ABB RobotStudio station: task2_Diaz_Raphael_good.rsstn

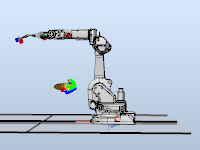
Station task2_Diaz_Raphael_good (saved by RobotStudio 7.0.8732.594)
Controller IRB_1660ID_4kg_1.55m_1
  mechanical unit ROB_1: IRB1660ID_4_155__03, 6 joints, base frame (0, 0, 0) mm
Layout (positions relative to the parent item):
  - IRB1660ID_4_155__03 [mechanism, from Robots\IRB1660ID_4_155__03.rslib] at (0, 0, 0) mm; joint values [0, 0, 0, 0, 0, 0] (rad or m)
  - Binzel_ID_22 [mechanism, from Tools\Binzel_ID_22.rslib] at (962.96, 0, 1296.5) mm, rotated rx 0 ry 90 rz 0 deg
  - propeller [part, from Training Objects\propeller.rslib] at (600, 300, 492) mm
Attachment: Binzel_ID_22 is attached to IRB1660ID_4_155__03 / Link6
Collision set Jeu de collisions_1: propeller against Binzel_ID_22, near miss 0.01 m
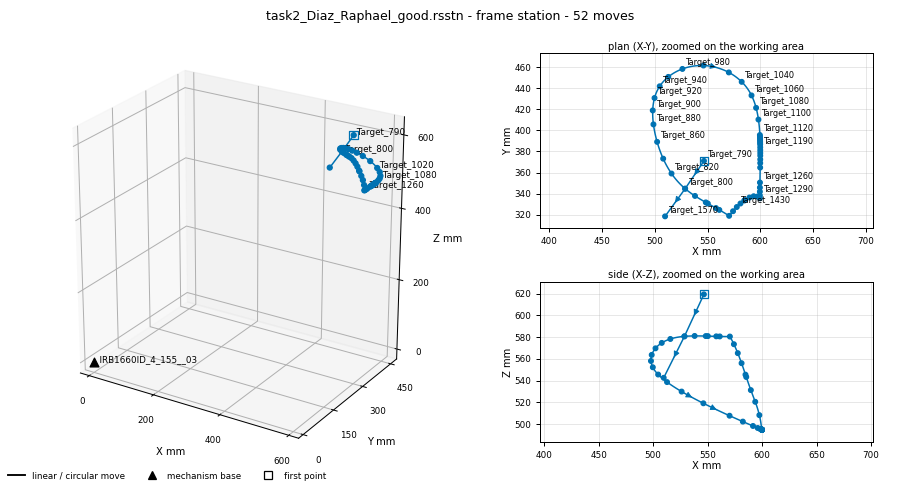
[picture p0: tool path of task2_Diaz_Raphael_good.rsstn in frame station, 52 of 54 moves have a stored position in this frame; points joined in program order, loops and branches not executed]
Targets, tools, work objects and paths stored in the station, written as RAPID:
! task T_ROB1
MODULE CalibData
  PERS tooldata tWeldGun:=[TRUE,[[49.841566361,0,372.194826196],[0.981627183,0,0.190808995,0]],[2,[0,0,100],[0,1,0,0],0,0,0]];
  TASK PERS wobjdata wobjpropeller:=[FALSE,TRUE,"",[[600,300,492],[1,0,0,0]],[[0,0,0],[1,0,0,0]]];
ENDMODULE

! task T_ROB1
MODULE Module1
  CONST robtarget Target_10:=[[-91.457935103,19.381495894,50.577643768],[0.33610531,0.650809481,-0.678295692,0.058268297],[0,0,0,0],[9E+09,9E+09,9E+09,9E+09,9E+09,9E+09]];
  CONST robtarget Target_20:=[[-71.308296548,44.654165227,88.72583181],[0.299329258,0.383053383,-0.856704989,0.172420021],[0,0,0,0],[9E+09,9E+09,9E+09,9E+09,9E+09,9E+09]];
  CONST robtarget Target_30:=[[-78.37226907,51.547933238,87.786349051],[0.117055584,0.822479759,0.470472306,-0.297457301],[0,0,0,0],[9E+09,9E+09,9E+09,9E+09,9E+09,9E+09]];
  CONST robtarget Target_40:=[[-84.2413284,59.034723416,86.319213476],[0.026567482,0.682501524,0.663067393,-0.306312701],[0,0,0,0],[9E+09,9E+09,9E+09,9E+09,9E+09,9E+09]];
  CONST robtarget Target_50:=[[-88.689736644,66.246127572,84.593004406],[0.015778406,-0.605999209,-0.736035915,0.301275841],[0,0,0,0],[9E+09,9E+09,9E+09,9E+09,9E+09,9E+09]];
  CONST robtarget Target_60:=[[-92.125721625,73.134318692,82.720919892],[0.04515113,-0.547999882,-0.781238502,0.29550619],[0,0,0,0],[9E+09,9E+09,9E+09,9E+09,9E+09,9E+09]];
  CONST robtarget Target_70:=[[-95.368783045,81.204603576,80.298199397],[0.073925684,-0.486542001,-0.821345688,0.288449537],[0,0,0,0],[9E+09,9E+09,9E+09,9E+09,9E+09,9E+09]];
  CONST robtarget Target_80:=[[-97.881197354,89.077633701,77.728399267],[0.099335356,-0.428105921,-0.853147584,0.281064062],[0,0,0,0],[9E+09,9E+09,9E+09,9E+09,9E+09,9E+09]];
  CONST robtarget Target_90:=[[-100.033550677,97.806160497,74.661081462],[0.123258623,-0.370832778,-0.879360143,0.272059003],[0,0,0,0],[9E+09,9E+09,9E+09,9E+09,9E+09,9E+09]];
  CONST robtarget Target_100:=[[-101.370571802,105.645030719,71.694531974],[0.137199941,-0.339206789,-0.892353586,0.264234759],[0,0,0,0],[9E+09,9E+09,9E+09,9E+09,9E+09,9E+09]];
  CONST robtarget Target_110:=[[-101.985517598,112.196954226,69.035342228],[0.143656337,-0.327575869,-0.897345121,0.25851236],[0,0,0,0],[9E+09,9E+09,9E+09,9E+09,9E+09,9E+09]];
  CONST robtarget Target_120:=[[-102.050783732,118.905008267,66.110246882],[0.145775207,-0.329044052,-0.897889581,0.253522978],[0,0,0,0],[9E+09,9E+09,9E+09,9E+09,9E+09,9E+09]];
  CONST robtarget Target_130:=[[-101.533339164,124.816905053,63.325398927],[0.144182461,-0.340855073,-0.894813654,0.249675314],[0,0,0,0],[9E+09,9E+09,9E+09,9E+09,9E+09,9E+09]];
  CONST robtarget Target_140:=[[-100.353288111,130.675770651,60.324888075],[0.139634307,-0.361631976,-0.888364776,0.246033736],[0,0,0,0],[9E+09,9E+09,9E+09,9E+09,9E+09,9E+09]];
  CONST robtarget Target_150:=[[-98.373944468,136.376977106,57.10491509],[0.132520307,-0.390029479,-0.878439143,0.242198359],[0,0,0,0],[9E+09,9E+09,9E+09,9E+09,9E+09,9E+09]];
  CONST robtarget Target_160:=[[-95.443552762,141.799075074,53.663228181],[0.123926919,-0.422628209,-0.865746717,0.23771861],[0,0,0,0],[9E+09,9E+09,9E+09,9E+09,9E+09,9E+09]];
  CONST robtarget Target_170:=[[-91.477533598,146.819277823,50.007346793],[0.119671198,-0.442406606,-0.857808795,0.232635489],[0,0,0,0],[9E+09,9E+09,9E+09,9E+09,9E+09,9E+09]];
  CONST robtarget Target_180:=[[-87.281413645,150.715782558,46.72049795],[0.119661723,-0.448819982,-0.855661661,0.228220987],[0,0,0,0],[9E+09,9E+09,9E+09,9E+09,9E+09,9E+09]];
  CONST robtarget Target_190:=[[-80.620544648,155.184469083,42.151881558],[0.123978964,-0.4449886,-0.858578449,0.222390219],[0,0,0,0],[9E+09,9E+09,9E+09,9E+09,9E+09,9E+09]];
  CONST robtarget Target_200:=[[-73.893581114,158.264895339,38.018756325],[0.131604396,-0.430683265,-0.866049681,0.217140869],[0,0,0,0],[9E+09,9E+09,9E+09,9E+09,9E+09,9E+09]];
  CONST robtarget Target_210:=[[-64.220289368,160.829182326,32.592775118],[0.147131247,-0.395863657,-0.88192952,0.209391221],[0,0,0,0],[9E+09,9E+09,9E+09,9E+09,9E+09,9E+09]];
  CONST robtarget Target_220:=[[-53.911152598,161.491173917,27.246893168],[0.169941176,-0.339310055,-0.903559757,0.198918197],[0,0,0,0],[9E+09,9E+09,9E+09,9E+09,9E+09,9E+09]];
  CONST robtarget Target_230:=[[-41.810424561,159.659563045,21.355681333],[0.200569217,-0.259415196,-0.927008519,0.182019097],[0,0,0,0],[9E+09,9E+09,9E+09,9E+09,9E+09,9E+09]];
  CONST robtarget Target_240:=[[-29.865399659,154.942077691,15.837356936],[0.23576805,-0.163069983,-0.945025663,0.157315299],[0,0,0,0],[9E+09,9E+09,9E+09,9E+09,9E+09,9E+09]];
  CONST robtarget Target_250:=[[-23.746821381,151.136846643,13.101781769],[0.258743132,-0.097071717,-0.951106966,0.137929734],[0,0,0,0],[9E+09,9E+09,9E+09,9E+09,9E+09,9E+09]];
  CONST robtarget Target_260:=[[-17.666404877,146.023270878,10.434303465],[0.288578567,-0.007433268,-0.951293254,0.108204906],[0,0,0,0],[9E+09,9E+09,9E+09,9E+09,9E+09,9E+09]];
  CONST robtarget Target_270:=[[-12.651720819,140.244931337,8.266059989],[0.323388208,0.102706042,-0.938405879,0.065314172],[0,0,0,0],[9E+09,9E+09,9E+09,9E+09,9E+09,9E+09]];
  CONST robtarget Target_280:=[[-8.342471887,133.132300705,6.417634315],[0.365484893,0.241842337,-0.898844698,-0.003359375],[0,0,0,0],[9E+09,9E+09,9E+09,9E+09,9E+09,9E+09]];
  CONST robtarget Target_290:=[[-5.860288763,127.302609884,5.357964601],[0.392577974,0.330559163,-0.856027592,-0.061886481],[0,0,0,0],[9E+09,9E+09,9E+09,9E+09,9E+09,9E+09]];
  CONST robtarget Target_300:=[[-3.992732838,121.340092984,4.564472039],[0.414682372,0.398212956,-0.809177456,-0.12123043],[0,0,0,0],[9E+09,9E+09,9E+09,9E+09,9E+09,9E+09]];
  CONST robtarget Target_310:=[[-2.622802171,115.344004565,3.985624159],[0.432618645,0.446096603,-0.762723965,-0.179139837],[0,0,0,0],[9E+09,9E+09,9E+09,9E+09,9E+09,9E+09]];
  CONST robtarget Target_320:=[[-1.767059875,110.242020204,3.626183876],[0.445232804,0.473650463,-0.725447966,-0.22615976],[0,0,0,0],[9E+09,9E+09,9E+09,9E+09,9E+09,9E+09]];
  CONST robtarget Target_330:=[[-0.982577099,103.57416667,3.298978191],[0.458683869,0.49524232,-0.681313145,-0.283119323],[0,0,0,0],[9E+09,9E+09,9E+09,9E+09,9E+09,9E+09]];
  CONST robtarget Target_340:=[[-0.419164603,95.575819275,3.066095193],[0.470824783,0.505758987,-0.636794178,-0.342089236],[0,0,0,0],[9E+09,9E+09,9E+09,9E+09,9E+09,9E+09]];
  CONST robtarget Target_350:=[[-0.347305784,94.031887162,3.036532706],[0.472698308,0.506466011,-0.629402289,-0.35199609],[0,0,0,0],[9E+09,9E+09,9E+09,9E+09,9E+09,9E+09]];
  CONST robtarget Target_360:=[[-0.286087854,92.508600465,3.011348256],[0.474402212,0.506869723,-0.622525025,-0.361231531],[0,0,0,0],[9E+09,9E+09,9E+09,9E+09,9E+09,9E+09]];
  CONST robtarget Target_370:=[[-0.23439904,91.006691049,2.990058478],[0.475942955,0.507030195,-0.616165129,-0.369782665],[0,0,0,0],[9E+09,9E+09,9E+09,9E+09,9E+09,9E+09]];
  CONST robtarget Target_380:=[[-0.191127564,89.526890776,2.972180009],[0.477327032,0.507002401,-0.610324314,-0.377639647],[0,0,0,0],[9E+09,9E+09,9E+09,9E+09,9E+09,9E+09]];
  CONST robtarget Target_390:=[[-0.155200515,88.069901279,2.957246513],[0.478560799,0.506836069,-0.605003836,-0.384794905],[0,0,0,0],[9E+09,9E+09,9E+09,9E+09,9E+09,9E+09]];
  CONST robtarget Target_400:=[[-0.125712724,86.636254313,2.944866369],[0.47965026,0.506575668,-0.600205327,-0.391241979],[0,0,0,0],[9E+09,9E+09,9E+09,9E+09,9E+09,9E+09]];
  CONST robtarget Target_410:=[[-0.08261427,83.840896172,2.926280967],[0.481425707,0.505921465,-0.592147985,-0.402036719],[0,0,0,0],[9E+09,9E+09,9E+09,9E+09,9E+09,9E+09]];
  CONST robtarget Target_420:=[[-0.056032781,81.142526543,2.913966515],[0.482919894,0.505164577,-0.585071946,-0.411446161],[0,0,0,0],[9E+09,9E+09,9E+09,9E+09,9E+09,9E+09]];
  CONST robtarget Target_430:=[[-0.043048917,78.537720407,2.906816995],[0.484257027,0.504334678,-0.578448423,-0.420165547],[0,0,0,0],[9E+09,9E+09,9E+09,9E+09,9E+09,9E+09]];
  CONST robtarget Target_440:=[[-0.0411167,76.022616297,2.903894485],[0.485444308,0.50348214,-0.572280664,-0.428187343],[0,0,0,0],[9E+09,9E+09,9E+09,9E+09,9E+09,9E+09]];
  CONST robtarget Target_450:=[[-0.054549222,72.411596474,2.905814438],[0.486961818,0.502254961,-0.563882455,-0.43891311],[0,0,0,0],[9E+09,9E+09,9E+09,9E+09,9E+09,9E+09]];
  CONST robtarget Target_460:=[[-0.082166755,68.986528626,2.913297006],[0.488190694,0.501190902,-0.556485739,-0.448108412],[0,0,0,0],[9E+09,9E+09,9E+09,9E+09,9E+09,9E+09]];
  CONST robtarget Target_470:=[[-0.131718126,64.695350259,2.928466957],[0.489437258,0.500158131,-0.54809675,-0.458129859],[0,0,0,0],[9E+09,9E+09,9E+09,9E+09,9E+09,9E+09]];
  CONST robtarget Target_480:=[[-0.336493102,50.490109414,2.996479603],[0.49131632,0.501098619,-0.528226501,-0.478001266],[0,0,0,0],[9E+09,9E+09,9E+09,9E+09,9E+09,9E+09]];
  CONST robtarget Target_490:=[[-0.389538706,45.718395544,3.014646231],[0.491239016,0.503319057,-0.524352335,-0.480009151],[0,0,0,0],[9E+09,9E+09,9E+09,9E+09,9E+09,9E+09]];
  CONST robtarget Target_500:=[[-0.416651037,41.829820629,3.023974096],[0.490943622,0.505849897,-0.522175178,-0.480024296],[0,0,0,0],[9E+09,9E+09,9E+09,9E+09,9E+09,9E+09]];
  CONST robtarget Target_510:=[[-0.425239936,38.15628616,3.026910604],[0.490487838,0.508788687,-0.520869322,-0.478801528],[0,0,0,0],[9E+09,9E+09,9E+09,9E+09,9E+09,9E+09]];
  CONST robtarget Target_520:=[[-0.41907447,35.554875844,3.024714783],[0.490068794,0.511158358,-0.520350237,-0.477268625],[0,0,0,0],[9E+09,9E+09,9E+09,9E+09,9E+09,9E+09]];
  CONST robtarget Target_530:=[[-1.239353828,36.579195021,10.094804089],[0.485285471,0.505393808,-0.570570399,-0.428397631],[0,0,0,0],[9E+09,9E+09,9E+09,9E+09,9E+09,9E+09]];
  CONST robtarget Target_540:=[[-2.503019666,37.269792356,16.365865608],[0.479926257,0.507544354,-0.597699632,-0.393477656],[0,0,0,0],[9E+09,9E+09,9E+09,9E+09,9E+09,9E+09]];
  CONST robtarget Target_550:=[[-4.236986629,37.619005876,22.65445378],[0.472203187,0.526252128,-0.609551252,-0.358510975],[0,0,0,0],[9E+09,9E+09,9E+09,9E+09,9E+09,9E+09]];
  CONST robtarget Target_560:=[[-6.286575332,37.504452968,28.619621674],[0.462621307,0.570105136,-0.592015985,-0.332383415],[0,0,0,0],[9E+09,9E+09,9E+09,9E+09,9E+09,9E+09]];
  CONST robtarget Target_570:=[[-8.20610761,37.063247875,33.701409225],[0.453744324,0.629847272,-0.535614332,-0.332454193],[0,0,0,0],[9E+09,9E+09,9E+09,9E+09,9E+09,9E+09]];
  CONST robtarget Target_580:=[[-10.318626049,36.285780987,39.360011182],[0.4392884,0.703953672,-0.435520626,-0.348993861],[0,0,0,0],[9E+09,9E+09,9E+09,9E+09,9E+09,9E+09]];
  CONST robtarget Target_590:=[[-12.661310127,35.078889502,45.926428415],[0.411372895,0.780339138,-0.279004478,-0.379472886],[0,0,0,0],[9E+09,9E+09,9E+09,9E+09,9E+09,9E+09]];
  CONST robtarget Target_600:=[[-14.532992973,33.887723981,51.407083874],[0.377332955,0.820678051,-0.122575,-0.411196725],[0,0,0,0],[9E+09,9E+09,9E+09,9E+09,9E+09,9E+09]];
  CONST robtarget Target_610:=[[-10.798566102,36.060475375,40.678801419],[0.563334326,0.293280069,-0.772407011,0.005352333],[0,0,-2,0],[9E+09,9E+09,9E+09,9E+09,9E+09,9E+09]];
  CONST robtarget Target_620:=[[-17.018667911,32.078049469,58.829591721],[0.549464464,0.601489484,-0.578324534,-0.042894489],[0,0,0,0],[9E+09,9E+09,9E+09,9E+09,9E+09,9E+09]];
  CONST robtarget Target_630:=[[-18.838902409,30.609710668,64.071754814],[0.530289122,0.699136232,-0.471191576,-0.089333504],[0,0,0,0],[9E+09,9E+09,9E+09,9E+09,9E+09,9E+09]];
  CONST robtarget Target_640:=[[-20.744338327,28.895776947,69.241801524],[0.123477381,0.8147616,-0.542306034,-0.163771293],[0,0,0,0],[9E+09,9E+09,9E+09,9E+09,9E+09,9E+09]];
  CONST robtarget Target_650:=[[-22.309539778,27.279666365,73.303790841],[0.110236403,0.855139822,-0.430096695,-0.267582985],[0,0,0,0],[9E+09,9E+09,9E+09,9E+09,9E+09,9E+09]];
  CONST robtarget Target_660:=[[-23.973327026,25.503693293,77.244247794],[0.470774997,0.638586467,-0.601652731,0.09269422],[0,0,0,0],[9E+09,9E+09,9E+09,9E+09,9E+09,9E+09]];
  CONST robtarget Target_670:=[[-25.872608406,23.295941961,81.501586218],[0.457862129,0.733090582,-0.501721122,0.034876705],[0,0,0,0],[9E+09,9E+09,9E+09,9E+09,9E+09,9E+09]];
  CONST robtarget Target_680:=[[-27.702454631,21.186772281,85.158169778],[0.001522806,-0.45137891,-0.779666651,0.434021512],[0,0,0,0],[9E+09,9E+09,9E+09,9E+09,9E+09,9E+09]];
  CONST robtarget Target_690:=[[-29.579108704,18.917792453,88.550574629],[0.047769483,-0.396812931,-0.828772501,0.391655098],[0,0,0,0],[9E+09,9E+09,9E+09,9E+09,9E+09,9E+09]];
  CONST robtarget Target_700:=[[-34.181159805,21.772283678,88.563733649],[0.00902881,-0.455561574,-0.785071733,0.419576581],[0,0,0,0],[9E+09,9E+09,9E+09,9E+09,9E+09,9E+09]];
  CONST robtarget Target_710:=[[-38.892044155,24.513127262,88.646240796],[0.005175513,0.466142387,0.770169888,-0.435342202],[0,0,0,0],[9E+09,9E+09,9E+09,9E+09,9E+09,9E+09]];
  CONST robtarget Target_720:=[[-42.068819563,26.298976235,88.725674008],[0.008188854,0.465500607,0.767643082,-0.440415969],[0,0,0,0],[9E+09,9E+09,9E+09,9E+09,9E+09,9E+09]];
  CONST robtarget Target_730:=[[-49.791866469,30.580230673,88.941782186],[0.000167691,-0.452797516,-0.778146204,0.435273324],[0,0,0,0],[9E+09,9E+09,9E+09,9E+09,9E+09,9E+09]];
  CONST robtarget Target_740:=[[-51.709318387,31.655936915,88.990570919],[0.0053493,-0.447245007,-0.783953208,0.430535315],[0,0,0,0],[9E+09,9E+09,9E+09,9E+09,9E+09,9E+09]];
  CONST robtarget Target_750:=[[-57.377839054,34.942502242,89.094223182],[0.02849914,-0.420022979,-0.809203176,0.409827666],[0,0,0,0],[9E+09,9E+09,9E+09,9E+09,9E+09,9E+09]];
  CONST robtarget Target_760:=[[-61.957234754,37.792717573,89.103595138],[0.059645275,-0.371858872,-0.84212475,0.385991355],[0,0,0,0],[9E+09,9E+09,9E+09,9E+09,9E+09,9E+09]];
  CONST robtarget Target_770:=[[-66.351329922,40.79265749,89.011564709],[0.115406616,-0.253755157,-0.893913867,0.351009446],[0,0,0,0],[9E+09,9E+09,9E+09,9E+09,9E+09,9E+09]];
  CONST robtarget Target_780:=[[-71.308296548,44.654165227,88.72583181],[0.299329258,0.383053383,-0.856704989,0.172420021],[0,0,0,0],[9E+09,9E+09,9E+09,9E+09,9E+09,9E+09]];
  CONST robtarget Target_790:=[[-53.446490384,71.034227347,127.305248995],[0.33610531,0.650809481,-0.678295692,0.058268297],[0,0,0,0],[9E+09,9E+09,9E+09,9E+09,9E+09,9E+09]];
  CONST robtarget Target_800:=[[-71.308296548,44.654165227,88.72583181],[0.33610531,0.650809481,-0.678295692,0.058268297],[0,0,0,0],[9E+09,9E+09,9E+09,9E+09,9E+09,9E+09]];
  CONST robtarget Target_810:=[[-78.37226907,51.547933238,87.786349051],[0.33610531,0.650809481,-0.678295692,0.058268297],[0,0,0,0],[9E+09,9E+09,9E+09,9E+09,9E+09,9E+09]];
  CONST robtarget Target_820:=[[-84.2413284,59.034723416,86.319213476],[0.33610531,0.650809481,-0.678295692,0.058268297],[0,0,0,0],[9E+09,9E+09,9E+09,9E+09,9E+09,9E+09]];
  CONST robtarget Target_830:=[[-88.689736644,66.246127572,84.593004406],[0.33610531,0.650809481,-0.678295692,0.058268297],[0,0,0,0],[9E+09,9E+09,9E+09,9E+09,9E+09,9E+09]];
  CONST robtarget Target_840:=[[-92.125721625,73.134318692,82.720919892],[0.33610531,0.650809481,-0.678295692,0.058268297],[0,0,0,0],[9E+09,9E+09,9E+09,9E+09,9E+09,9E+09]];
  CONST robtarget Target_850:=[[-95.368783045,81.204603576,80.298199397],[0.33610531,0.650809481,-0.678295692,0.058268297],[0,0,0,0],[9E+09,9E+09,9E+09,9E+09,9E+09,9E+09]];
  CONST robtarget Target_860:=[[-97.881197354,89.077633701,77.728399267],[0.33610531,0.650809481,-0.678295692,0.058268297],[0,0,0,0],[9E+09,9E+09,9E+09,9E+09,9E+09,9E+09]];
  CONST robtarget Target_870:=[[-100.033550677,97.806160497,74.661081462],[0.33610531,0.650809481,-0.678295692,0.058268297],[0,0,0,0],[9E+09,9E+09,9E+09,9E+09,9E+09,9E+09]];
  CONST robtarget Target_880:=[[-101.370571802,105.645030719,71.694531974],[0.33610531,0.650809481,-0.678295692,0.058268297],[0,0,0,0],[9E+09,9E+09,9E+09,9E+09,9E+09,9E+09]];
  CONST robtarget Target_890:=[[-101.985517598,112.196954226,69.035342228],[0.33610531,0.650809481,-0.678295692,0.058268297],[0,0,0,0],[9E+09,9E+09,9E+09,9E+09,9E+09,9E+09]];
  CONST robtarget Target_900:=[[-102.050783732,118.905008267,66.110246882],[0.33610531,0.650809481,-0.678295692,0.058268297],[0,0,0,0],[9E+09,9E+09,9E+09,9E+09,9E+09,9E+09]];
  CONST robtarget Target_910:=[[-101.533339164,124.816905053,63.325398927],[0.33610531,0.650809481,-0.678295692,0.058268297],[0,0,0,0],[9E+09,9E+09,9E+09,9E+09,9E+09,9E+09]];
  CONST robtarget Target_920:=[[-100.353288111,130.675770651,60.324888075],[0.33610531,0.650809481,-0.678295692,0.058268297],[0,0,0,0],[9E+09,9E+09,9E+09,9E+09,9E+09,9E+09]];
  CONST robtarget Target_930:=[[-98.373944468,136.376977106,57.10491509],[0.33610531,0.650809481,-0.678295692,0.058268297],[0,0,0,0],[9E+09,9E+09,9E+09,9E+09,9E+09,9E+09]];
  CONST robtarget Target_940:=[[-95.443552762,141.799075074,53.663228181],[0.33610531,0.650809481,-0.678295692,0.058268297],[0,0,0,0],[9E+09,9E+09,9E+09,9E+09,9E+09,9E+09]];
  CONST robtarget Target_950:=[[-91.477533598,146.819277823,50.007346793],[0.33610531,0.650809481,-0.678295692,0.058268297],[0,0,0,0],[9E+09,9E+09,9E+09,9E+09,9E+09,9E+09]];
  CONST robtarget Target_960:=[[-87.281413645,150.715782558,46.72049795],[0.33610531,0.650809481,-0.678295692,0.058268297],[0,0,0,0],[9E+09,9E+09,9E+09,9E+09,9E+09,9E+09]];
  CONST robtarget Target_970:=[[-80.620544648,155.184469083,42.151881558],[0.33610531,0.650809481,-0.678295692,0.058268297],[0,0,0,0],[9E+09,9E+09,9E+09,9E+09,9E+09,9E+09]];
  CONST robtarget Target_980:=[[-73.893581114,158.264895339,38.018756325],[0.33610531,0.650809481,-0.678295692,0.058268297],[0,0,0,0],[9E+09,9E+09,9E+09,9E+09,9E+09,9E+09]];
  CONST robtarget Target_990:=[[-64.220289368,160.829182326,32.592775118],[0.33610531,0.650809481,-0.678295692,0.058268297],[0,0,0,0],[9E+09,9E+09,9E+09,9E+09,9E+09,9E+09]];
  CONST robtarget Target_1000:=[[-53.911152598,161.491173917,27.246893168],[0.33610531,0.650809481,-0.678295692,0.058268297],[0,0,0,0],[9E+09,9E+09,9E+09,9E+09,9E+09,9E+09]];
  CONST robtarget Target_1010:=[[-41.810424561,159.659563045,21.355681333],[0.33610531,0.650809481,-0.678295692,0.058268297],[0,0,0,0],[9E+09,9E+09,9E+09,9E+09,9E+09,9E+09]];
  CONST robtarget Target_1020:=[[-29.865399659,154.942077691,15.837356936],[0.33610531,0.650809481,-0.678295692,0.058268297],[0,0,0,0],[9E+09,9E+09,9E+09,9E+09,9E+09,9E+09]];
  CONST robtarget Target_1030:=[[-23.746821381,151.136846643,13.101781769],[0.33610531,0.650809481,-0.678295692,0.058268297],[0,0,0,0],[9E+09,9E+09,9E+09,9E+09,9E+09,9E+09]];
  CONST robtarget Target_1040:=[[-17.666404877,146.023270878,10.434303465],[0.33610531,0.650809481,-0.678295692,0.058268297],[0,0,0,0],[9E+09,9E+09,9E+09,9E+09,9E+09,9E+09]];
  CONST robtarget Target_1050:=[[-12.651720819,140.244931337,8.266059989],[0.33610531,0.650809481,-0.678295692,0.058268297],[0,0,0,0],[9E+09,9E+09,9E+09,9E+09,9E+09,9E+09]];
  CONST robtarget Target_1060:=[[-8.342471887,133.132300705,6.417634315],[0.33610531,0.650809481,-0.678295692,0.058268297],[0,0,0,0],[9E+09,9E+09,9E+09,9E+09,9E+09,9E+09]];
  CONST robtarget Target_1070:=[[-5.860288763,127.302609884,5.357964601],[0.33610531,0.650809481,-0.678295692,0.058268297],[0,0,0,0],[9E+09,9E+09,9E+09,9E+09,9E+09,9E+09]];
  CONST robtarget Target_1080:=[[-3.992732838,121.340092984,4.564472039],[0.33610531,0.650809481,-0.678295692,0.058268297],[0,0,0,0],[9E+09,9E+09,9E+09,9E+09,9E+09,9E+09]];
  CONST robtarget Target_1090:=[[-2.622802171,115.344004565,3.985624159],[0.33610531,0.650809481,-0.678295692,0.058268297],[0,0,0,0],[9E+09,9E+09,9E+09,9E+09,9E+09,9E+09]];
  CONST robtarget Target_1100:=[[-1.767059875,110.242020204,3.626183876],[0.33610531,0.650809481,-0.678295692,0.058268297],[0,0,0,0],[9E+09,9E+09,9E+09,9E+09,9E+09,9E+09]];
  CONST robtarget Target_1110:=[[-0.982577099,103.57416667,3.298978191],[0.33610531,0.650809481,-0.678295692,0.058268297],[0,0,0,0],[9E+09,9E+09,9E+09,9E+09,9E+09,9E+09]];
  CONST robtarget Target_1120:=[[-0.419164603,95.575819275,3.066095193],[0.33610531,0.650809481,-0.678295692,0.058268297],[0,0,0,0],[9E+09,9E+09,9E+09,9E+09,9E+09,9E+09]];
  CONST robtarget Target_1130:=[[-0.347305784,94.031887162,3.036532706],[0.33610531,0.650809481,-0.678295692,0.058268297],[0,0,0,0],[9E+09,9E+09,9E+09,9E+09,9E+09,9E+09]];
  CONST robtarget Target_1140:=[[-0.286087854,92.508600465,3.011348256],[0.33610531,0.650809481,-0.678295692,0.058268297],[0,0,0,0],[9E+09,9E+09,9E+09,9E+09,9E+09,9E+09]];
  CONST robtarget Target_1150:=[[-0.23439904,91.006691049,2.990058478],[0.33610531,0.650809481,-0.678295692,0.058268297],[0,0,0,0],[9E+09,9E+09,9E+09,9E+09,9E+09,9E+09]];
  CONST robtarget Target_1160:=[[-0.191127564,89.526890776,2.972180009],[0.33610531,0.650809481,-0.678295692,0.058268297],[0,0,0,0],[9E+09,9E+09,9E+09,9E+09,9E+09,9E+09]];
  CONST robtarget Target_1170:=[[-0.155200515,88.069901279,2.957246513],[0.33610531,0.650809481,-0.678295692,0.058268297],[0,0,0,0],[9E+09,9E+09,9E+09,9E+09,9E+09,9E+09]];
  CONST robtarget Target_1180:=[[-0.125712724,86.636254313,2.944866369],[0.33610531,0.650809481,-0.678295692,0.058268297],[0,0,0,0],[9E+09,9E+09,9E+09,9E+09,9E+09,9E+09]];
  CONST robtarget Target_1190:=[[-0.08261427,83.840896172,2.926280967],[0.33610531,0.650809481,-0.678295692,0.058268297],[0,0,0,0],[9E+09,9E+09,9E+09,9E+09,9E+09,9E+09]];
  CONST robtarget Target_1200:=[[-0.056032781,81.142526543,2.913966515],[0.33610531,0.650809481,-0.678295692,0.058268297],[0,0,0,0],[9E+09,9E+09,9E+09,9E+09,9E+09,9E+09]];
  CONST robtarget Target_1210:=[[-0.043048917,78.537720407,2.906816995],[0.33610531,0.650809481,-0.678295692,0.058268297],[0,0,0,0],[9E+09,9E+09,9E+09,9E+09,9E+09,9E+09]];
  CONST robtarget Target_1220:=[[-0.0411167,76.022616297,2.903894485],[0.33610531,0.650809481,-0.678295692,0.058268297],[0,0,0,0],[9E+09,9E+09,9E+09,9E+09,9E+09,9E+09]];
  CONST robtarget Target_1230:=[[-0.054549222,72.411596474,2.905814438],[0.33610531,0.650809481,-0.678295692,0.058268297],[0,0,0,0],[9E+09,9E+09,9E+09,9E+09,9E+09,9E+09]];
  CONST robtarget Target_1240:=[[-0.082166755,68.986528626,2.913297006],[0.33610531,0.650809481,-0.678295692,0.058268297],[0,0,0,0],[9E+09,9E+09,9E+09,9E+09,9E+09,9E+09]];
  CONST robtarget Target_1250:=[[-0.131718126,64.695350259,2.928466957],[0.33610531,0.650809481,-0.678295692,0.058268297],[0,0,0,0],[9E+09,9E+09,9E+09,9E+09,9E+09,9E+09]];
  CONST robtarget Target_1260:=[[-0.336493102,50.490109414,2.996479603],[0.33610531,0.650809481,-0.678295692,0.058268297],[0,0,0,0],[9E+09,9E+09,9E+09,9E+09,9E+09,9E+09]];
  CONST robtarget Target_1270:=[[-0.389538706,45.718395544,3.014646231],[0.33610531,0.650809481,-0.678295692,0.058268297],[0,0,0,0],[9E+09,9E+09,9E+09,9E+09,9E+09,9E+09]];
  CONST robtarget Target_1280:=[[-0.416651037,41.829820629,3.023974096],[0.33610531,0.650809481,-0.678295692,0.058268297],[0,0,0,0],[9E+09,9E+09,9E+09,9E+09,9E+09,9E+09]];
  CONST robtarget Target_1290:=[[-0.425239936,38.15628616,3.026910604],[0.33610531,0.650809481,-0.678295692,0.058268297],[0,0,0,0],[9E+09,9E+09,9E+09,9E+09,9E+09,9E+09]];
  CONST robtarget Target_1300:=[[-0.41907447,35.554875844,3.024714783],[0.33610531,0.650809481,-0.678295692,0.058268297],[0,0,0,0],[9E+09,9E+09,9E+09,9E+09,9E+09,9E+09]];
  CONST robtarget Target_1310:=[[-1.239353828,36.579195021,10.094804089],[0.33610531,0.650809481,-0.678295692,0.058268297],[0,0,0,0],[9E+09,9E+09,9E+09,9E+09,9E+09,9E+09]];
  CONST robtarget Target_1320:=[[-2.503019666,37.269792356,16.365865608],[0.33610531,0.650809481,-0.678295692,0.058268297],[0,0,0,0],[9E+09,9E+09,9E+09,9E+09,9E+09,9E+09]];
  CONST robtarget Target_1330:=[[-4.236986629,37.619005876,22.65445378],[0.33610531,0.650809481,-0.678295692,0.058268297],[0,0,0,0],[9E+09,9E+09,9E+09,9E+09,9E+09,9E+09]];
  CONST robtarget Target_1340:=[[-6.286575332,37.504452968,28.619621674],[0.33610531,0.650809481,-0.678295692,0.058268297],[0,0,0,0],[9E+09,9E+09,9E+09,9E+09,9E+09,9E+09]];
  CONST robtarget Target_1350:=[[-8.20610761,37.063247875,33.701409225],[0.33610531,0.650809481,-0.678295692,0.058268297],[0,0,0,0],[9E+09,9E+09,9E+09,9E+09,9E+09,9E+09]];
  CONST robtarget Target_1360:=[[-10.318626049,36.285780987,39.360011182],[0.33610531,0.650809481,-0.678295692,0.058268297],[0,0,0,0],[9E+09,9E+09,9E+09,9E+09,9E+09,9E+09]];
  CONST robtarget Target_1370:=[[-12.661310127,35.078889502,45.926428415],[0.33610531,0.650809481,-0.678295692,0.058268297],[0,0,0,0],[9E+09,9E+09,9E+09,9E+09,9E+09,9E+09]];
  CONST robtarget Target_1380:=[[-14.532992973,33.887723981,51.407083874],[0.33610531,0.650809481,-0.678295692,0.058268297],[0,0,0,0],[9E+09,9E+09,9E+09,9E+09,9E+09,9E+09]];
  CONST robtarget Target_1390:=[[-15.252203225,33.390108645,53.548500087],[0.33610531,0.650809481,-0.678295692,0.058268297],[0,0,0,0],[9E+09,9E+09,9E+09,9E+09,9E+09,9E+09]];
  CONST robtarget Target_1400:=[[-17.018667911,32.078049469,58.829591721],[0.33610531,0.650809481,-0.678295692,0.058268297],[0,0,0,0],[9E+09,9E+09,9E+09,9E+09,9E+09,9E+09]];
  CONST robtarget Target_1410:=[[-18.838902409,30.609710668,64.071754814],[0.33610531,0.650809481,-0.678295692,0.058268297],[0,0,0,0],[9E+09,9E+09,9E+09,9E+09,9E+09,9E+09]];
  CONST robtarget Target_1420:=[[-20.744338327,28.895776947,69.241801524],[0.33610531,0.650809481,-0.678295692,0.058268297],[0,0,0,0],[9E+09,9E+09,9E+09,9E+09,9E+09,9E+09]];
  CONST robtarget Target_1430:=[[-22.309539778,27.279666365,73.303790841],[0.33610531,0.650809481,-0.678295692,0.058268297],[0,0,0,0],[9E+09,9E+09,9E+09,9E+09,9E+09,9E+09]];
  CONST robtarget Target_1440:=[[-23.973327026,25.503693293,77.244247794],[0.33610531,0.650809481,-0.678295692,0.058268297],[0,0,0,0],[9E+09,9E+09,9E+09,9E+09,9E+09,9E+09]];
  CONST robtarget Target_1450:=[[-25.872608406,23.295941961,81.501586218],[0.33610531,0.650809481,-0.678295692,0.058268297],[0,0,0,0],[9E+09,9E+09,9E+09,9E+09,9E+09,9E+09]];
  CONST robtarget Target_1460:=[[-27.702454631,21.186772281,85.158169778],[0.33610531,0.650809481,-0.678295692,0.058268297],[0,0,0,0],[9E+09,9E+09,9E+09,9E+09,9E+09,9E+09]];
  CONST robtarget Target_1470:=[[-29.579108704,18.917792453,88.550574629],[0.33610531,0.650809481,-0.678295692,0.058268297],[0,0,0,0],[9E+09,9E+09,9E+09,9E+09,9E+09,9E+09]];
  CONST robtarget Target_1480:=[[-34.181159805,21.772283678,88.563733649],[0.33610531,0.650809481,-0.678295692,0.058268297],[0,0,0,0],[9E+09,9E+09,9E+09,9E+09,9E+09,9E+09]];
  CONST robtarget Target_1490:=[[-38.892044155,24.513127262,88.646240796],[0.33610531,0.650809481,-0.678295692,0.058268297],[0,0,0,0],[9E+09,9E+09,9E+09,9E+09,9E+09,9E+09]];
  CONST robtarget Target_1500:=[[-42.068819563,26.298976235,88.725674008],[0.33610531,0.650809481,-0.678295692,0.058268297],[0,0,0,0],[9E+09,9E+09,9E+09,9E+09,9E+09,9E+09]];
  CONST robtarget Target_1510:=[[-49.791866469,30.580230673,88.941782186],[0.33610531,0.650809481,-0.678295692,0.058268297],[0,0,0,0],[9E+09,9E+09,9E+09,9E+09,9E+09,9E+09]];
  CONST robtarget Target_1520:=[[-51.709318387,31.655936915,88.990570919],[0.33610531,0.650809481,-0.678295692,0.058268297],[0,0,0,0],[9E+09,9E+09,9E+09,9E+09,9E+09,9E+09]];
  CONST robtarget Target_1530:=[[-57.377839054,34.942502242,89.094223182],[0.33610531,0.650809481,-0.678295692,0.058268297],[0,0,0,0],[9E+09,9E+09,9E+09,9E+09,9E+09,9E+09]];
  CONST robtarget Target_1540:=[[-61.957234754,37.792717573,89.103595138],[0.33610531,0.650809481,-0.678295692,0.058268297],[0,0,0,0],[9E+09,9E+09,9E+09,9E+09,9E+09,9E+09]];
  CONST robtarget Target_1550:=[[-66.351329922,40.79265749,89.011564709],[0.33610531,0.650809481,-0.678295692,0.058268297],[0,0,0,0],[9E+09,9E+09,9E+09,9E+09,9E+09,9E+09]];
  CONST robtarget Target_1560:=[[-71.308296548,44.654165227,88.72583181],[0.33610531,0.650809481,-0.678295692,0.058268297],[0,0,0,0],[9E+09,9E+09,9E+09,9E+09,9E+09,9E+09]];
  CONST robtarget Target_1570:=[[-90.346612088,18.416300625,50.658562371],[0.33610531,0.650809481,-0.678295692,0.058268297],[0,0,0,0],[9E+09,9E+09,9E+09,9E+09,9E+09,9E+09]];
  CONST jointtarget JtHome_1:=[[0,0,0,0,0,0],[9E+09,9E+09,9E+09,9E+09,9E+09,9E+09]];
  PROC Path_10()
    MoveJ Target_790,v3000,z1,tWeldGun\WObj:=wobjpropeller;
    MoveL Target_800,v300,z1,tWeldGun\WObj:=wobjpropeller;
    MoveC Target_810,Target_820,v300,z1,tWeldGun\WObj:=wobjpropeller;
    MoveC Target_830,Target_840,v300,z1,tWeldGun\WObj:=wobjpropeller;
    MoveC Target_850,Target_860,v300,z1,tWeldGun\WObj:=wobjpropeller;
    MoveC Target_870,Target_880,v300,z1,tWeldGun\WObj:=wobjpropeller;
    MoveC Target_890,Target_900,v300,z1,tWeldGun\WObj:=wobjpropeller;
    MoveC Target_910,Target_920,v300,z1,tWeldGun\WObj:=wobjpropeller;
    MoveC Target_930,Target_940,v300,z1,tWeldGun\WObj:=wobjpropeller;
    MoveC Target_950,Target_960,v300,z1,tWeldGun\WObj:=wobjpropeller;
    MoveC Target_970,Target_980,v300,z1,tWeldGun\WObj:=wobjpropeller;
    MoveC Target_990,Target_1000,v300,z1,tWeldGun\WObj:=wobjpropeller;
    MoveC Target_1010,Target_1020,v300,z1,tWeldGun\WObj:=wobjpropeller;
    MoveC Target_1030,Target_1040,v300,z1,tWeldGun\WObj:=wobjpropeller;
    MoveC Target_1050,Target_1060,v300,z1,tWeldGun\WObj:=wobjpropeller;
    MoveC Target_1070,Target_1080,v300,z1,tWeldGun\WObj:=wobjpropeller;
    MoveC Target_1090,Target_1100,v300,z1,tWeldGun\WObj:=wobjpropeller;
    MoveC Target_1110,Target_1120,v300,z1,tWeldGun\WObj:=wobjpropeller;
    MoveL Target_1130,v300,z1,tWeldGun\WObj:=wobjpropeller;
    MoveL Target_1140,v300,z1,tWeldGun\WObj:=wobjpropeller;
    MoveL Target_1150,v300,z1,tWeldGun\WObj:=wobjpropeller;
    MoveL Target_1160,v300,z1,tWeldGun\WObj:=wobjpropeller;
    MoveL Target_1170,v300,z1,tWeldGun\WObj:=wobjpropeller;
    MoveL Target_1180,v300,z1,tWeldGun\WObj:=wobjpropeller;
    MoveL Target_1190,v300,z1,tWeldGun\WObj:=wobjpropeller;
    MoveL Target_1200,v300,z1,tWeldGun\WObj:=wobjpropeller;
    MoveL Target_1210,v300,z1,tWeldGun\WObj:=wobjpropeller;
    MoveL Target_1220,v300,z1,tWeldGun\WObj:=wobjpropeller;
    MoveL Target_1230,v300,z1,tWeldGun\WObj:=wobjpropeller;
    MoveL Target_1240,v300,z1,tWeldGun\WObj:=wobjpropeller;
    MoveL Target_1250,v300,z1,tWeldGun\WObj:=wobjpropeller;
    MoveL Target_1260,v300,z1,tWeldGun\WObj:=wobjpropeller;
    MoveL Target_1270,v300,z1,tWeldGun\WObj:=wobjpropeller;
    MoveL Target_1280,v300,z1,tWeldGun\WObj:=wobjpropeller;
    MoveL Target_1290,v300,z1,tWeldGun\WObj:=wobjpropeller;
    MoveL Target_1300,v300,z1,tWeldGun\WObj:=wobjpropeller;
    MoveC Target_1310,Target_1320,v300,z1,tWeldGun\WObj:=wobjpropeller;
    MoveC Target_1330,Target_1340,v300,z1,tWeldGun\WObj:=wobjpropeller;
    MoveC Target_1350,Target_1360,v300,z1,tWeldGun\WObj:=wobjpropeller;
    MoveC Target_1370,Target_1380,v300,z1,tWeldGun\WObj:=wobjpropeller;
    MoveL Target_1390,v300,z1,tWeldGun\WObj:=wobjpropeller;
    MoveC Target_1400,Target_1410,v300,z1,tWeldGun\WObj:=wobjpropeller;
    MoveC Target_1420,Target_1430,v300,z1,tWeldGun\WObj:=wobjpropeller;
    MoveC Target_1440,Target_1450,v300,z1,tWeldGun\WObj:=wobjpropeller;
    MoveC Target_1460,Target_1470,v300,z1,tWeldGun\WObj:=wobjpropeller;
    MoveC Target_1480,Target_1490,v300,z1,tWeldGun\WObj:=wobjpropeller;
    MoveL Target_1500,v300,z1,tWeldGun\WObj:=wobjpropeller;
    MoveL Target_1510,v300,z1,tWeldGun\WObj:=wobjpropeller;
    MoveL Target_1520,v300,z1,tWeldGun\WObj:=wobjpropeller;
    MoveC Target_1530,Target_1540,v300,z1,tWeldGun\WObj:=wobjpropeller;
    MoveC Target_1550,Target_1560,v300,z1,tWeldGun\WObj:=wobjpropeller;
    MoveL Target_1570,v300,z1,tWeldGun\WObj:=wobjpropeller;
  ENDPROC
  PROC main()
    MoveAbsJ JtHome_1,v1000,z100,tWeldGun\WObj:=wobjpropeller;
    Path_10;
    MoveAbsJ JtHome_1,v1000,z100,tWeldGun\WObj:=wobjpropeller;
  ENDPROC
ENDMODULE

